Fanuc TP program (LS listing): ENTER2ZONE.LS

/PROG  ENTER2ZONE
/ATTR
OWNER		= MNEDITOR;
COMMENT		= "";
PROG_SIZE	= 320;
CREATE		= DATE 11-05-20  TIME 11:03:02;
MODIFIED	= DATE 11-06-15  TIME 17:57:16;
FILE_NAME	= ENTER2ZO;
VERSION		= 0;
LINE_COUNT	= 3;
MEMORY_SIZE	= 728;
PROTECT		= READ;
TCD:  STACK_SIZE	= 0,
      TASK_PRIORITY	= 50,
      TIME_SLICE	= 0,
      BUSY_LAMP_OFF	= 0,
      ABORT_REQUEST	= 0,
      PAUSE_REQUEST	= 0;
DEFAULT_GROUP	= *,*,*,*,*;
CONTROL_CODE	= 00000000 00000000;
/APPL
/APPL
  SPOT : TRUE ;
/MN
   1:  CALL MREQZONE(9,16,9999999) ;
   2:  WAIT $MASY_GRP[1].$OK_ENTER=1    ;
   3:  CALL MGETZONE(2,16,9999999) ;
/POS
/END
